// TIA Portal V19 export
TYPE "EFC_STATUS_WORD"
   STRUCT
      ErrorCode0 : Bool := false;
      ErrorCode1 : Bool := false;
      ErrorCode2 : Bool := false;
      ErrorCode3 : Bool := false;
      ErrorCode4 : Bool := false;
      ErrorCode5 : Bool := false;
      ErrorCode6 : Bool := false;
      ErrorCode7 : Bool := false;
      Reverse : Bool := false;
      Running : Bool := false;
      Jogging : Bool := false;
      Accelerating : Bool := false;
      Decelerating : Bool := false;
      OverVoltage : Bool := false;
      OverCurrent : Bool := false;
      Error : Bool := false;
   END_STRUCT;
END_TYPE
